// TIA Portal V19 export
DATA_BLOCK "MixingIngredientsApplePie"   // DB225
// stored: MemoryReserve 100
   VAR
      mixingApplePie { S7_SetPoint := 'True'} : "typeMixingIngredientsPieApple";
   END_VAR
BEGIN
END_DATA_BLOCK
